FUNCTION_BLOCK FB_2CAM_SelectCameraMap
VAR_INPUT

	bMap2x5:					BOOL;

	stPackCamera1Map2x5		: ST_SCANNER_CameraMap;
	stPackCamera2Map2x5		: ST_SCANNER_CameraMap;
END_VAR
VAR_OUTPUT
	stPackCamera1Map		: ST_SCANNER_CameraMap;
	stPackCamera2Map		: ST_SCANNER_CameraMap;
END_VAR
VAR
END_VAR

IF bMap2x5 THEN
	stPackCamera1Map := stPackCamera1Map2x5;
	stPackCamera2Map := stPackCamera2Map2x5;
END_IF

END_FUNCTION_BLOCK

(* stored: Version 1.1.0.1, ProductVersion 3.1.4024.15
   POU FB_2CAM_SelectCameraMap: Id {3fe82204-90f8-46d5-8e73-20a78e044f6f}, SpecialFunc None *)
